// TIA Portal V19 export
DATA_BLOCK "PPrf_MAIN"   // DB96
{ DB_Accessible_From_OPC_UA := 'FALSE' }
// stored: Access Published, DBAccessibleFromOPCUA false, MemoryReserve 100
   VAR RETAIN
      PIVOT : Array[1.."PPRF_TOTAL_ARCHIVE_ITEMS"] of "Prg_Pivot";
   END_VAR
   VAR
      GET_ITF : "Prg_GetITF";
      RWD : Struct
         EMPTY { ExternalAccessible := 'False'; ExternalVisible := 'False'; ExternalWritable := 'False'} : "PPrf_Data";
         UPDATE { ExternalAccessible := 'False'; ExternalVisible := 'False'; ExternalWritable := 'False'} : "PPrf_Data";
         GET { ExternalAccessible := 'False'; ExternalVisible := 'False'; ExternalWritable := 'False'} : "PPrf_Data";
         HMI : "PPrf_Data";
         SCADA : "PPrf_Data";
      END_STRUCT;
      HMI : "Prg_HMI";
      SCADA : "Prg_SCADA";
   END_VAR
   VAR RETAIN
      ON_WORK : "PPrf_Data";
   END_VAR
BEGIN
END_DATA_BLOCK
